// TIA Portal V20 export
DATA_BLOCK "ET500SP_501"   // DB228
// stored: MemoryReserve 100
   VAR
      "SP501.00 CONTROL DC POWER TRIPPED E156CB" : Bool;
      "SP501.01 SAFETY DC POWER TRIPPED E218CB" : Bool;
      SPARE1 : Bool;
      SPARE2 : Bool;
      "SP501.04 Vision STO" : Bool;
      "SP501.05 Vision Judgment" : Bool;
      SPARE3 : Bool;
      SPARE4 : Bool;
      SPARE5 : Bool;
      SPARE6 : Bool;
      SPARE7 : Bool;
      SPARE8 : Bool;
      SPARE9 : Bool;
      SPARE10 : Bool;
      SPARE11 : Bool;
      SPARE12 : Bool;
   END_VAR
BEGIN
END_DATA_BLOCK
